(* PLC project Unnamed, Unknown Unnamed 1 *)
(* stored: creationDateTime 2022-12-13T19:44:02, modificationDateTime 2022-12-19T12:41:08 *)

PROGRAM water_tank
  VAR
    Start AT %IX0.0 : BOOL := 0;
    Stop AT %IX0.1 : BOOL := 1;
    High AT %IX0.2 : BOOL;
    Low AT %IX0.3 : BOOL;
    Height AT %IW0 : UINT;
    High_Limit AT %IW1 : UINT;
    Low_Limit AT %IW2 : UINT;
    Master AT %IX0.4 : BOOL;
    Valve_In AT %QX0.0 : BOOL;
    Valve_Out AT %QX0.1 : BOOL;
  END_VAR

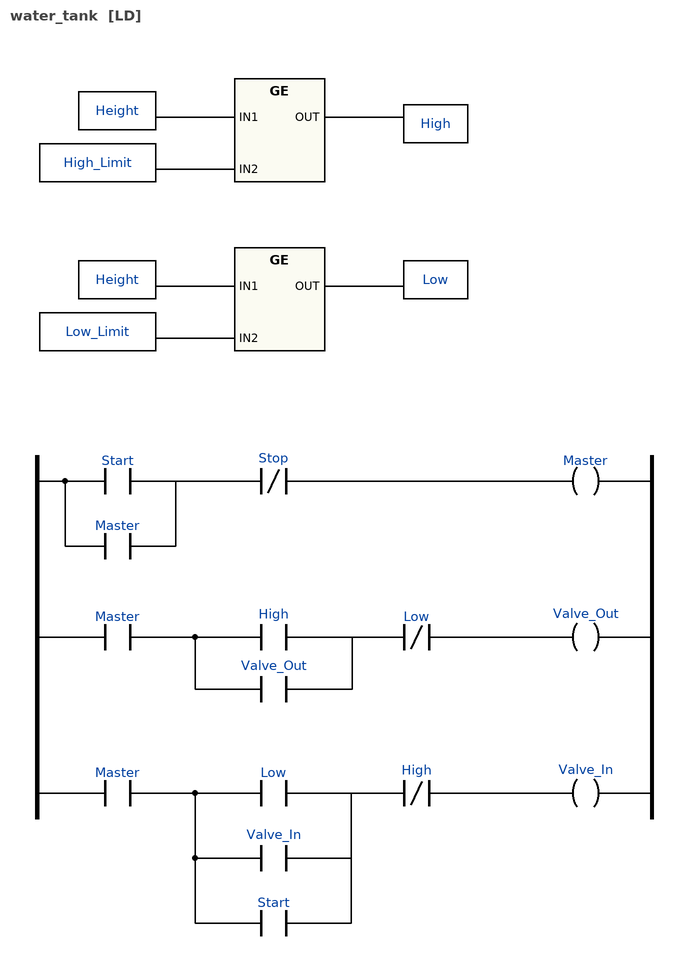
(* LD diagram, written out as Structured Text *)
High := Height >= High_Limit;
Low := Height >= Low_Limit;
Master := (Start OR Master) AND NOT Stop;
Valve_Out := Master AND (High OR Valve_Out) AND NOT Low;
Valve_In := Master AND (Low OR Valve_In OR Start) AND NOT High;
END_PROGRAM

CONFIGURATION Config0
  RESOURCE Res0 ON PLC
    TASK task0(INTERVAL := T#20ms, PRIORITY := 0);
    PROGRAM instance0 WITH task0 : water_tank;
  END_RESOURCE
END_CONFIGURATION
